TYPE ST_EP3751_HMI EXTENDS ST_HmiFunction :
	STRUCT
		// Unit in 1G
		ACC_X : REAL;
		ACC_Y : REAL;
		ACC_Z : REAL;
		// °/s
		Gyro_X : REAL;
		Gyro_Y : REAL;
		Gyro_Z : REAL;
		// Angles
		Roll  : REAL;
		Pitch : REAL;
	END_STRUCT
END_TYPE

(* stored: Version 1.1.0.1
   DUT ST_EP3751_HMI: Id {65fe18cb-7c8d-4002-abf2-b6d1cb347281} *)
